# EPICS substitutions: example.substitutions
# SPDX-FileCopyrightText: 2006 Argonne National Laboratory
#
# SPDX-License-Identifier: EPICS

# Example substitutions file

file "db/circle.db" {
	{ user = "${USER}" }
}

file "db/dbExample1.db" {
	{ user = "${USER}" }
}

file db/dbExample2.db {
	pattern { user, no, scan }
		{ "${USER}", 1, "1 second" }
		{ "${USER}", 2, "2 second" }
		{ "${USER}", 3, "5 second" }
}
